(* LS Electric XG5000 project: XMC_LSDedicated_FBs *)
(* sample programs for LS dedicated  function blocks. *)
(* PLC LSPLC *)
(* module base 0 slot 0: Input/Output Module:XMC-DN24 (DC 24V Input 8Points/TR output 16Points) *)
(* module base 0 slot 1: Internal Analog Input/Output:XMF-AH04E (A/D voltage/current 2 channels, D/A voltage 2 channels) *)
(* task Periodic Task: Kind=2 *)
(* task Initialization Task: Kind=1 *)
(* task NC Program: Kind=6 *)

PROGRAM ECAT_Connect_Example (* task: Scan Program *)
VAR
    Connect_Error : BOOL; (* status that LS_Connect has an error *)
    Connect_ErrorID : WORD; (* LS_Connect Error number *)
    Connect_INST : LS_CONNECT; (* LS_Connect fb *)
    Disconnect_Error : BOOL; (* status that LS_Disconnect has an error *)
    Disconnect_ErrorID : WORD; (* Error Number for LS_Disconnect FB *)
    Disconnect_INST : LS_DISCONNECT; (* LS_Disconnect fb *)
    Execute_Connect : BOOL; (* Execute LS_Connect fb *)
    Execute_Disconnect : BOOL; (* execute LS_Disconnect fb *)
END_VAR

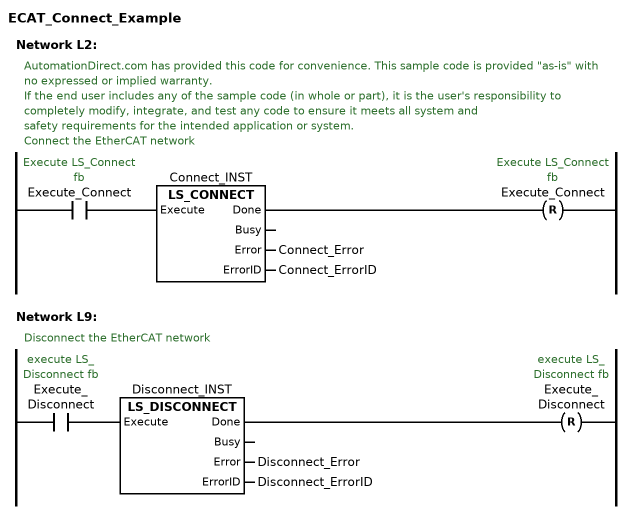
(* AutomationDirect.com has provided this code for convenience. This sample code is provided "as-is" with no expressed or implied warranty. / If the end user includes any of the sample code (in whole or part), it is the user's responsibility to completely modify, integrate, and test any code to ensure it meets all system and / safety requirements for the intended application or system. *)
(* Connect the EtherCAT network *)
(* Rung L2 *)
Connect_INST(Execute := Execute_Connect, Error => Connect_Error, ErrorID => Connect_ErrorID);
IF Connect_INST.Done THEN Execute_Connect := FALSE; END_IF;
(* Disconnect the EtherCAT network *)
(* Rung L9 *)
Disconnect_INST(Execute := Execute_Disconnect, Error => Disconnect_Error, ErrorID => Disconnect_ErrorID);
IF Disconnect_INST.Done THEN Execute_Disconnect := FALSE; END_IF;
END_PROGRAM

PROGRAM MC_PowerAll_Example (* task: Scan Program *)
(* example program for MC_PowerAll *)
VAR
    All_Axes_Ready : BOOL; (* flag that all axes are ready *)
    PowerAll_Error : BOOL; (* status of MC_Power error status *)
    PowerAll_ErrorID : WORD; (* error id of Axis 1 MC_Power *)
    PowerAll_INST : MC_POWERALL; (* MC_PowerALL fb *)
    PowerAll_Status : BOOL; (* status of axis 1 power *)
    PowerAll_Valid : BOOL; (* Axis1 power status is valid *)
    Power_On_Axis1 : BOOL; (* command to turn on power to axis 1 *)
END_VAR

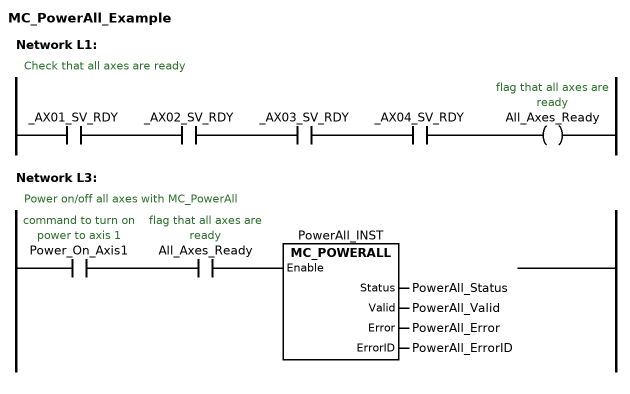
(* Check that all axes are ready *)
(* Rung L1 *)
All_Axes_Ready := _AX01_SV_RDY AND _AX02_SV_RDY AND _AX03_SV_RDY AND _AX04_SV_RDY;
(* Power on/off all axes with MC_PowerAll *)
(* Rung L3 *)
PowerAll_INST(Enable := Power_On_Axis1 AND All_Axes_Ready, Status => PowerAll_Status, Valid => PowerAll_Valid, Error => PowerAll_Error, ErrorID => PowerAll_ErrorID);
END_PROGRAM

PROGRAM Home_Example (* task: Scan Program *)
(* example of MC_Home and LS_Home *)
VAR
    All_Axes_Pwr_On : BOOL; (* status that all axes are powered on *)
    All_Axes_Ready : BOOL; (* flag that all axes are ready *)
    Execute_LS_HomeAll : BOOL; (* Execute LS_Home fb *)
    Execute_MC_HomeAll : BOOL; (* execute MC_Home fb *)
    LSHomeAll_Aborted : BOOL; (* LS_Home fb command aborted status *)
    LSHomeAll_Active : BOOL; (* LS_Home fb active status *)
    LSHomeAll_Busy : BOOL; (* LS_Home busy status *)
    LSHomeAll_Error : BOOL; (* LSHome fb error status *)
    LSHomeAll_ErrorID : WORD; (* LS_Home fb error id value *)
    LSHomeAll_INST : LS_HOMEALL; (* LS_HomeAll fb *)
    MCHomeAll_Aborted : BOOL; (* MC_Home command was aborted *)
    MCHomeAll_Active : BOOL; (* MC_Home is active *)
    MCHomeAll_Busy : BOOL; (* MC_Home is busy *)
    MCHomeAll_Error : BOOL; (* error status of MC_Home *)
    MCHomeAll_ErrorID : WORD; (* error id value for MC_Home *)
    MCHomeAll_INST : MC_HOMEALL; (* MC_HomeAll fb *)
END_VAR

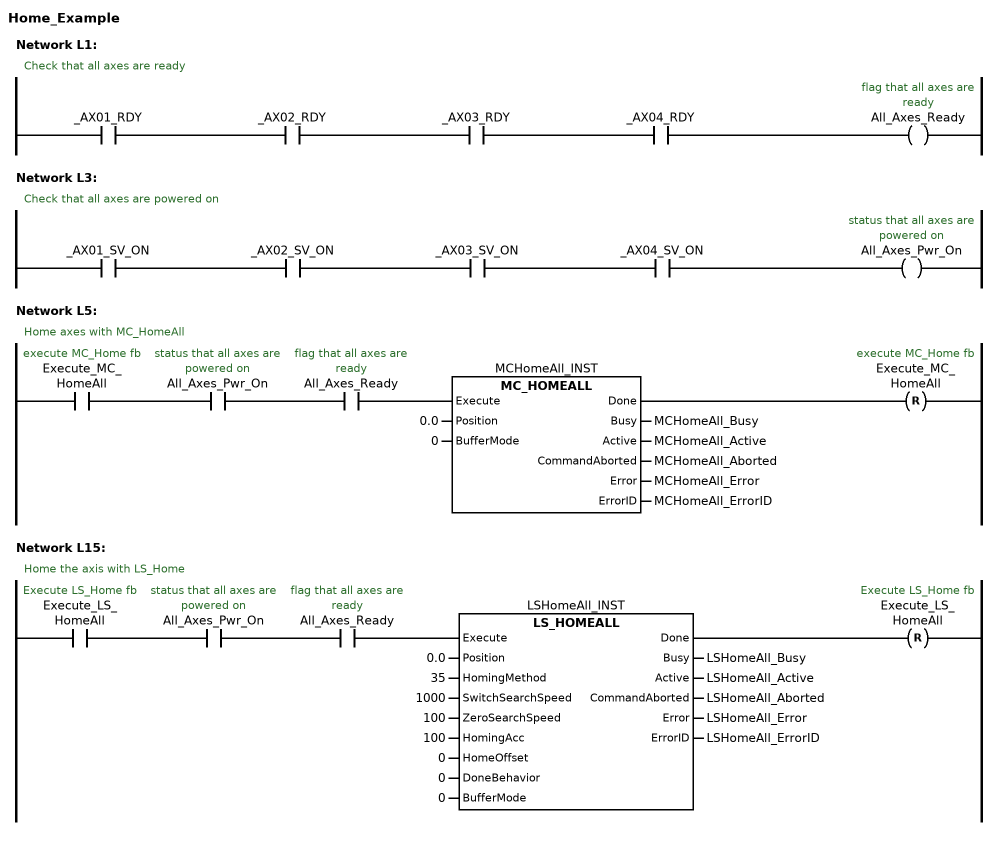
(* Check that all axes are ready *)
(* Rung L1 *)
All_Axes_Ready := _AX01_RDY AND _AX02_RDY AND _AX03_RDY AND _AX04_RDY;
(* Check that all axes are powered on *)
(* Rung L3 *)
All_Axes_Pwr_On := _AX01_SV_ON AND _AX02_SV_ON AND _AX03_SV_ON AND _AX04_SV_ON;
(* Home axes with MC_HomeAll *)
(* Rung L5 *)
MCHomeAll_INST(Execute := Execute_MC_HomeAll AND All_Axes_Pwr_On AND All_Axes_Ready, Position := 0.0, BufferMode := 0, Busy => MCHomeAll_Busy, Active => MCHomeAll_Active, CommandAborted => MCHomeAll_Aborted, Error => MCHomeAll_Error, ErrorID => MCHomeAll_ErrorID);
IF MCHomeAll_INST.Done THEN Execute_MC_HomeAll := FALSE; END_IF;
(* Home the axis with LS_Home *)
(* Rung L15 *)
LSHomeAll_INST(Execute := Execute_LS_HomeAll AND All_Axes_Pwr_On AND All_Axes_Ready, Position := 0.0, HomingMethod := 35, SwitchSearchSpeed := 1000, ZeroSearchSpeed := 100, HomingAcc := 100, HomeOffset := 0, DoneBehavior := 0, BufferMode := 0, Busy => LSHomeAll_Busy, Active => LSHomeAll_Active, CommandAborted => LSHomeAll_Aborted, Error => LSHomeAll_Error, ErrorID => LSHomeAll_ErrorID);
IF LSHomeAll_INST.Done THEN Execute_LS_HomeAll := FALSE; END_IF;
END_PROGRAM

PROGRAM MCStopAll_MCHaltAll_Examples (* task: Scan Program *)
(* Examples of MC_Stop and MC_Hault function blocks. *)
VAR
    All_Axes_Pwr_On : BOOL; (* status that all axes are powered on *)
    All_Axes_Ready : BOOL; (* flag that all axes are ready *)
    Execute_MCHaltAll : BOOL; (* execute MC_Halt FB *)
    Execute_MCStopAll : BOOL; (* command to execute MC_Stop fb *)
    MCHaltAll_Aborted : BOOL; (* MC_Hault command aborted status *)
    MCHaltAll_Active : BOOL; (* MC_Halt active status *)
    MCHaltAll_Busy : BOOL; (* Busy status for MC_Halt *)
    MCHaltAll_Error : BOOL; (* MC_Halt error status *)
    MCHaltAll_ErrorID : WORD; (* MC_Halt Error identification value *)
    MCHaltAll_INST : MC_HALTALL; (* MC_HaltAll fb *)
    MCStopAll_Aborted : BOOL; (* MC_Stop aborted status *)
    MCStopAll_Busy : BOOL; (* MC_Stop Busy Status *)
    MCStopAll_Error : BOOL; (* MC_Stop error status *)
    MCStopAll_ErrorID : WORD; (* MC_Stop error identification value *)
    MCStopAll_INST : MC_STOPALL; (* MC_Stop function block *)
END_VAR

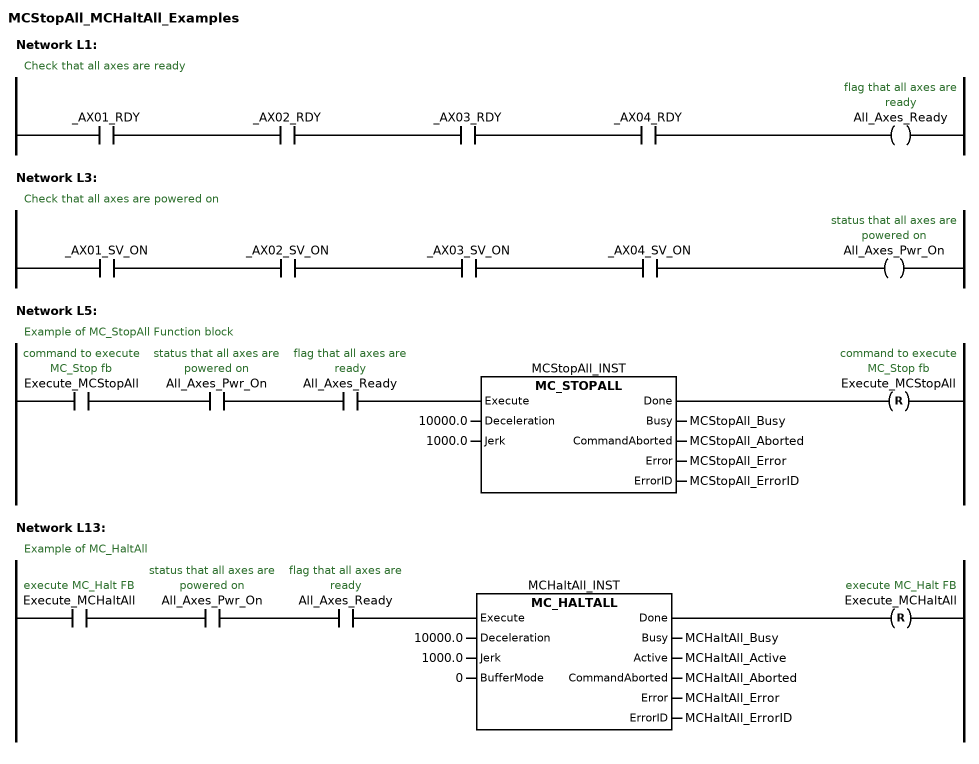
(* Check that all axes are ready *)
(* Rung L1 *)
All_Axes_Ready := _AX01_RDY AND _AX02_RDY AND _AX03_RDY AND _AX04_RDY;
(* Check that all axes are powered on *)
(* Rung L3 *)
All_Axes_Pwr_On := _AX01_SV_ON AND _AX02_SV_ON AND _AX03_SV_ON AND _AX04_SV_ON;
(* Example of MC_StopAll Function block *)
(* Rung L5 *)
MCStopAll_INST(Execute := Execute_MCStopAll AND All_Axes_Pwr_On AND All_Axes_Ready, Deceleration := 10000.0, Jerk := 1000.0, Busy => MCStopAll_Busy, CommandAborted => MCStopAll_Aborted, Error => MCStopAll_Error, ErrorID => MCStopAll_ErrorID);
IF MCStopAll_INST.Done THEN Execute_MCStopAll := FALSE; END_IF;
(* Example of MC_HaltAll *)
(* Rung L13 *)
MCHaltAll_INST(Execute := Execute_MCHaltAll AND All_Axes_Pwr_On AND All_Axes_Ready, Deceleration := 10000.0, Jerk := 1000.0, BufferMode := 0, Busy => MCHaltAll_Busy, Active => MCHaltAll_Active, CommandAborted => MCHaltAll_Aborted, Error => MCHaltAll_Error, ErrorID => MCHaltAll_ErrorID);
IF MCHaltAll_INST.Done THEN Execute_MCHaltAll := FALSE; END_IF;
END_PROGRAM

PROGRAM MC_Reset2All_Example (* task: Scan Program *)
(* example of MC_Reset2All function block. *)
VAR
    All_Axes_Ready : BOOL; (* flag that all axes are ready *)
    Execute_MCReset2All : BOOL; (* command to execute MC_Reset2 *)
    Reset2All_Busy : BOOL; (* busy status for MC_Reset2 *)
    Reset2All_Error : BOOL; (* error status for MC_Reset2 *)
    Reset2All_ErrorID : WORD; (* MC_Reset2 error identification *)
    Reset2All_ErrorType : UINT; (* error type for MC_Reset2 *)
    Reset2All_INST : MC_RESET2ALL; (* MC_Reset2All fb *)
END_VAR

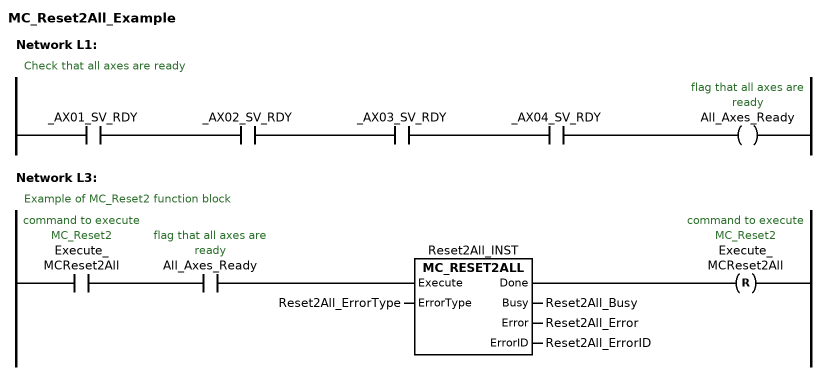
(* Check that all axes are ready *)
(* Rung L1 *)
All_Axes_Ready := _AX01_SV_RDY AND _AX02_SV_RDY AND _AX03_SV_RDY AND _AX04_SV_RDY;
(* Example of MC_Reset2 function block *)
(* Rung L3 *)
Reset2All_INST(Execute := Execute_MCReset2All AND All_Axes_Ready, ErrorType := Reset2All_ErrorType, Busy => Reset2All_Busy, Error => Reset2All_Error, ErrorID => Reset2All_ErrorID);
IF Reset2All_INST.Done THEN Execute_MCReset2All := FALSE; END_IF;
END_PROGRAM

PROGRAM LS_MoveLink_Example (* task: Scan Program *)
(* example of LS_MoveLink function block *)
VAR
    All_Axes_Pwr_On : BOOL; (* status that all axes are powered on *)
    All_Axes_Ready : BOOL; (* flag that all axes are ready *)
    Execute_MoveLink_Example : BOOL; (* execute the LS_MoveLink example *)
    Master_Axis : UINT; (* master axis of MC_CamIn *)
    MoveLink_Aborted : BOOL; (* aborted status for LS_MoveLink *)
    MoveLink_Active : BOOL; (* Active status for LS_MoveLink *)
    MoveLink_Busy : BOOL; (* busy status for LS_MoveLink *)
    MoveLink_Error : BOOL; (* error status for LS_MoveLink *)
    MoveLink_ErrorID : WORD; (* Error identification for LS_MoveLink *)
    MoveLink_INST : LS_MOVELINK; (* LS_MoveLink function block. *)
    MoveLink_InSync : BOOL; (* InSync status for LS_MoveLink *)
    MoveLink_MasterEndDistance : LREAL; (* MasterEndDistance for LS_MoveLink *)
    MoveLink_MasterStartDistance : LREAL; (* MasterStartDistance for LS_MoveLink *)
    MoveLink_MasterSyncPosition : LREAL; (* MasterSyncPosition for LS_MoveLink *)
    MoveLink_MasterValueSource : UINT; (* MasterValueSource for LS_MoveLink *)
    MoveLink_RatioDenominator : UDINT; (* RatioDenominator for LS_MoveLink *)
    MoveLink_RatioNumerator : DINT; (* RatioNumerator for LS_MoveLink *)
    MoveLink_SlaveEndPosition : LREAL; (* SlaveEndPosition for LS_MoveLink *)
    MoveLink_SlaveSyncPosition : LREAL; (* SlaveSyncPosition for LS_MoveLink *)
    MoveLink_SlaveWaitPosition : LREAL; (* SlaveWaitPosition for LS_MoveLink *)
    MoveLink_StartSync : BOOL; (* StartSync for LS_MoveLink *)
    MoveVelocity_INST : MC_MOVEVELOCITY; (* MC_MoveVelocity for master axis *)
    Slave_Axis : UINT; (* slave axis of MC_CamIn *)
END_VAR

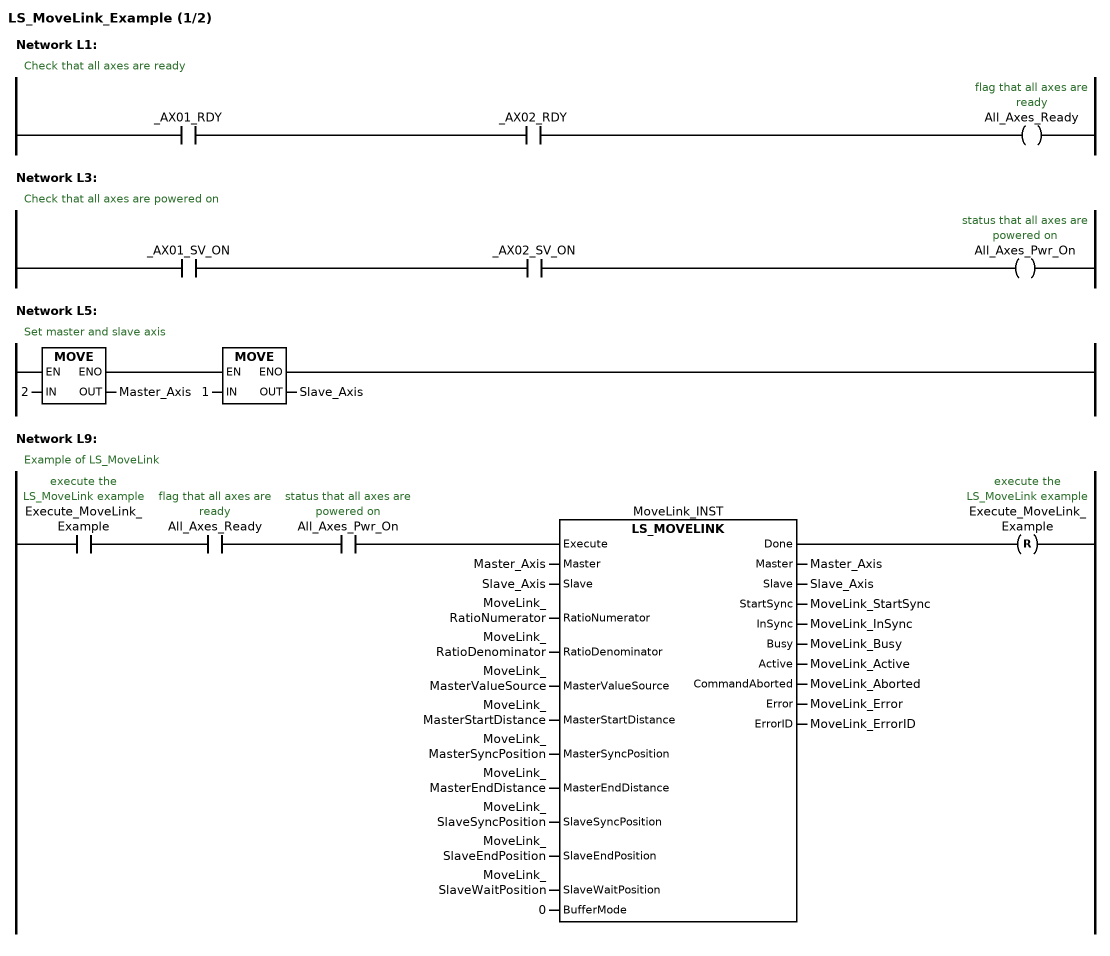
(* Check that all axes are ready *)
(* Rung L1 *)
All_Axes_Ready := _AX01_RDY AND _AX02_RDY;
(* Check that all axes are powered on *)
(* Rung L3 *)
All_Axes_Pwr_On := _AX01_SV_ON AND _AX02_SV_ON;
(* Set master and slave axis *)
(* Rung L5 *)
Master_Axis := 2;
Slave_Axis := 1;
(* Example of LS_MoveLink *)
(* Rung L9 *)
MoveLink_INST(Execute := Execute_MoveLink_Example AND All_Axes_Ready AND All_Axes_Pwr_On, Master := Master_Axis, Slave := Slave_Axis, RatioNumerator := MoveLink_RatioNumerator, RatioDenominator := MoveLink_RatioDenominator, MasterValueSource := MoveLink_MasterValueSource, MasterStartDistance := MoveLink_MasterStartDistance, MasterSyncPosition := MoveLink_MasterSyncPosition, MasterEndDistance := MoveLink_MasterEndDistance, SlaveSyncPosition := MoveLink_SlaveSyncPosition, SlaveEndPosition := MoveLink_SlaveEndPosition, SlaveWaitPosition := MoveLink_SlaveWaitPosition, BufferMode := 0, Master => Master_Axis, Slave => Slave_Axis, StartSync => MoveLink_StartSync, InSync => MoveLink_InSync, Busy => MoveLink_Busy, Active => MoveLink_Active, CommandAborted => MoveLink_Aborted, Error => MoveLink_Error, ErrorID => MoveLink_ErrorID);
IF MoveLink_INST.Done THEN Execute_MoveLink_Example := FALSE; END_IF;

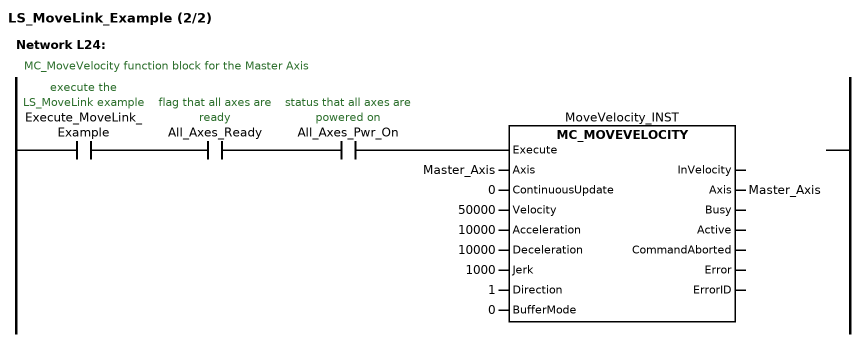
(* MC_MoveVelocity function block for the Master Axis *)
(* Rung L24 *)
MoveVelocity_INST(Execute := Execute_MoveLink_Example AND All_Axes_Ready AND All_Axes_Pwr_On, Axis := Master_Axis, ContinuousUpdate := 0, Velocity := 50000, Acceleration := 10000, Deceleration := 10000, Jerk := 1000, Direction := 1, BufferMode := 0, Axis => Master_Axis);
END_PROGRAM

PROGRAM LS_Jog_Example (* task: Scan Program *)
(* Example of LS_Jog function block. *)
VAR
    Axis1 : UINT; (* Variable for axis 1 *)
    Execute_FwdJog : BOOL; (* execute forward jog *)
    Execute_RevJog : BOOL; (* Execute reverse jog *)
    ForwardJog : LS_JOG; (* LS_Jog function block for forward jog *)
    FWD_Busy : BOOL; (* forward jog busy status *)
    FWD_Enabled : BOOL; (* forward jog enabled *)
    FWD_Error : BOOL; (* forward jog error status *)
    FWD_ErrorID : WORD; (* error identification for Forward jog *)
    FWD_Low_High : BOOL; (* low speed or high speed for forward jog *)
    ReverseJog : LS_JOG; (* LS_Jog for reverse jogging *)
    REV_Busy : BOOL; (* busy status for reverse jog *)
    REV_Enabled : BOOL; (* Enabled for reverse jog *)
    REV_Error : BOOL; (* error status for reverse jog *)
    REV_ErrorID : WORD; (* error identification for reverse jog *)
    REV_Low_High : BOOL; (* Low speed or high speed for reverse jog *)
END_VAR

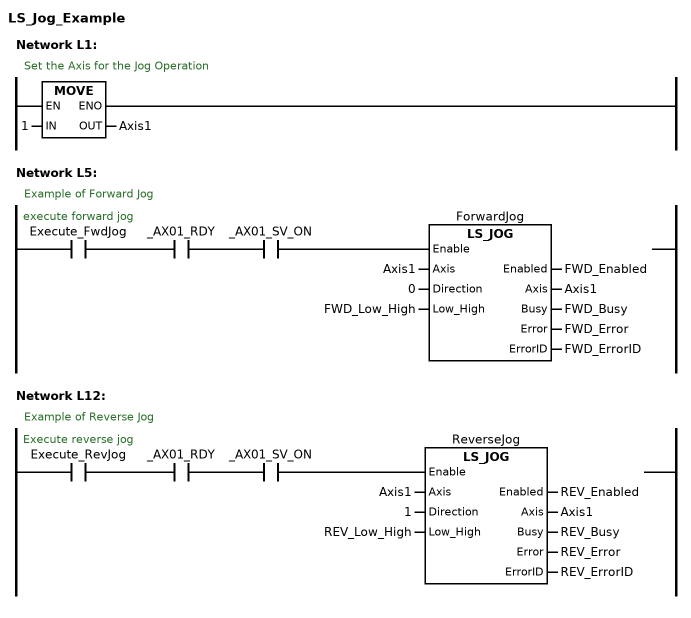
(* Set the Axis for the Jog Operation *)
(* Rung L1 *)
Axis1 := 1;
(* Example of Forward Jog *)
(* Rung L5 *)
ForwardJog(Enable := Execute_FwdJog AND _AX01_RDY AND _AX01_SV_ON, Axis := Axis1, Direction := 0, Low_High := FWD_Low_High, Enabled => FWD_Enabled, Axis => Axis1, Busy => FWD_Busy, Error => FWD_Error, ErrorID => FWD_ErrorID);
(* Example of Reverse Jog *)
(* Rung L12 *)
ReverseJog(Enable := Execute_RevJog AND _AX01_RDY AND _AX01_SV_ON, Axis := Axis1, Direction := 1, Low_High := REV_Low_High, Enabled => REV_Enabled, Axis => Axis1, Busy => REV_Busy, Error => REV_Error, ErrorID => REV_ErrorID);
END_PROGRAM

PROGRAM SDO_Operations (* task: Scan Program *)
(* example of LS_ReadSDO2, LS_WriteSDO2 and LS_SaveSDO *)
VAR
    Execute_ReadSDO : BOOL; (* command to execute LS_ReadSDO2 *)
    Execute_SaveSDO : BOOL; (* command to execute Save SDO on slave *)
    Execute_WriteSDO : BOOL; (* command to execute LS_WriteSDO2 *)
    ReadSDO_Busy : BOOL; (* Busy status for LS_ReadSDO2 *)
    ReadSDO_Error : BOOL; (* error status for LS_ReadSDO2 *)
    ReadSDO_ErrorID : WORD; (* error identification for LS_ReadSDO2 *)
    ReadSDO_Index : WORD; (* index to read from *)
    ReadSDO_INST : LS_READSDO2; (* LS_ReadSDO2 function block *)
    ReadSDO_Length : UINT; (* Length of data to read in bytes *)
    ReadSDO_Slave : UINT; (* Slave to read SDO *)
    ReadSDO_SubIndex : WORD; (* SubIndex to read *)
    ReadSDO_Value : DINT; (* value returned from SDO read *)
    SaveSDO_Busy : BOOL; (* busy status of LS_SaveSDO *)
    SaveSDO_Error : BOOL; (* Error status of LS_SaveSDO *)
    SaveSDO_ErrorID : WORD; (* error identification of LS_SaveSDO *)
    SaveSDO_INST : LS_SAVESDO; (* LS_SaveSDO function block *)
    SaveSDO_Slave : UINT; (* slave to save sdo *)
    WriteSDO_Busy : BOOL; (* busy status for LS_WriteSDO2 *)
    WriteSDO_Error : BOOL; (* Error Status for LS_WriteSDO2 *)
    WriteSDO_ErrorID : WORD; (* Error Identification for LS_WriteSDO2 *)
    WriteSDO_Index : WORD; (* Index to write to *)
    WriteSDO_INST : LS_WRITESDO2; (* LS_WriteSDO2 function block *)
    WriteSDO_Length : UINT; (* Length of data to write *)
    WriteSDO_Slave : UINT; (* slave to write SDO to *)
    WriteSDO_SubIndex : WORD; (* SubIndex to write to *)
    WriteSDO_Value : DINT; (* value to write to slave *)
END_VAR

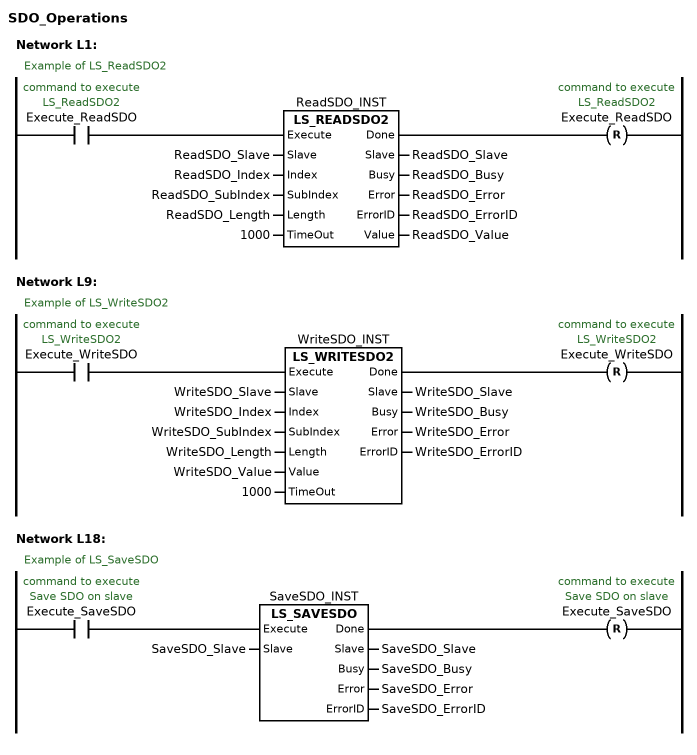
(* Example of LS_ReadSDO2 *)
(* Rung L1 *)
ReadSDO_INST(Execute := Execute_ReadSDO, Slave := ReadSDO_Slave, Index := ReadSDO_Index, SubIndex := ReadSDO_SubIndex, Length := ReadSDO_Length, TimeOut := 1000, Slave => ReadSDO_Slave, Busy => ReadSDO_Busy, Error => ReadSDO_Error, ErrorID => ReadSDO_ErrorID, Value => ReadSDO_Value);
IF ReadSDO_INST.Done THEN Execute_ReadSDO := FALSE; END_IF;
(* Example of LS_WriteSDO2 *)
(* Rung L9 *)
WriteSDO_INST(Execute := Execute_WriteSDO, Slave := WriteSDO_Slave, Index := WriteSDO_Index, SubIndex := WriteSDO_SubIndex, Length := WriteSDO_Length, Value := WriteSDO_Value, TimeOut := 1000, Slave => WriteSDO_Slave, Busy => WriteSDO_Busy, Error => WriteSDO_Error, ErrorID => WriteSDO_ErrorID);
IF WriteSDO_INST.Done THEN Execute_WriteSDO := FALSE; END_IF;
(* Example of LS_SaveSDO *)
(* Rung L18 *)
SaveSDO_INST(Execute := Execute_SaveSDO, Slave := SaveSDO_Slave, Slave => SaveSDO_Slave, Busy => SaveSDO_Busy, Error => SaveSDO_Error, ErrorID => SaveSDO_ErrorID);
IF SaveSDO_INST.Done THEN Execute_SaveSDO := FALSE; END_IF;
END_PROGRAM

PROGRAM LS_EncoderPreset_Example (* task: Scan Program *)
(* example of LS_EncoderPreset function block *)
VAR
    EncoderPreset_Busy : BOOL; (* busy status for LS_EncoderPreset *)
    EncoderPreset_Error : BOOL; (* error status for LS_EncoderPreset *)
    EncoderPreset_ErrorID : WORD; (* error identificaton for LS_EncoderPreset *)
    EncoderPreset_INST : LS_ENCODERPRESET; (* LS_EncoderPreset function block *)
    EncoderPreset_Position : LREAL; (* position to set encoder to *)
    EncoderPreset_Relative : BOOL; (* is position relative or absolute from current position *)
    EncoderToSet : UINT; (* choose the encoder value to change *)
    Execute_EncoderPreset : BOOL; (* execute the LS_EncoderPreset function block *)
END_VAR

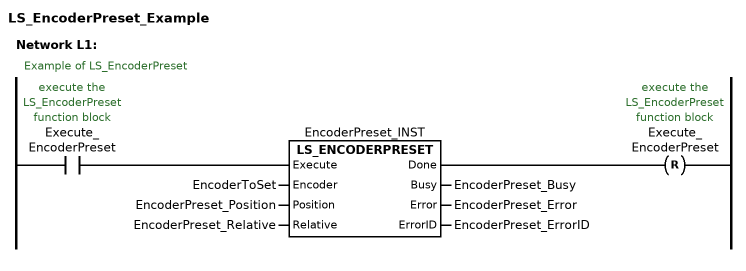
(* Example of LS_EncoderPreset *)
(* Rung L1 *)
EncoderPreset_INST(Execute := Execute_EncoderPreset, Encoder := EncoderToSet, Position := EncoderPreset_Position, Relative := EncoderPreset_Relative, Busy => EncoderPreset_Busy, Error => EncoderPreset_Error, ErrorID => EncoderPreset_ErrorID);
IF EncoderPreset_INST.Done THEN Execute_EncoderPreset := FALSE; END_IF;
END_PROGRAM